{attribute addProperty BoxType "EK1100-0000-0018"}
{attribute addProperty Id "Beckhoff_EPP4xxxEK1122Beckhoff_EPP4xxxEK1122_3C04EF3C1312164"}
{attribute addProperty CRC "990435394"}
{attribute addProperty SizeInBites "1312"}
{attribute addProperty SizeInBytes "164"}
TYPE Beckhoff_EPP4xxx_3B08D842 EXTENDS EK1100_179A0949 :
STRUCT
	{attribute addProperty Name "Beckhoff_EPP4xxxEK1122"}
	Beckhoff_EPP4xxxEK1122 : Beckhoff_EPP4xxxEK1122_3C04EF3C;
END_STRUCT
END_TYPE

(* stored: Version 1.2.0.0, ProductVersion 3.1.4024.9
   DUT Beckhoff_EPP4xxx_3B08D842: Id {6dd08b7d-8ac4-4a50-8f7f-34f95e6a53e4} *)
